// TIA Portal V19 export
DATA_BLOCK "IO-LinkDevicesDB"   // DB210
VERSION : 0.0
// stored: AutoNumber false, InstanceOfName IO-Link Devices, InstanceOfType FB
"IO-Link Devices"
   // VAR
   //    PNIODiag : Struct
   //       StationOK : Bool;
   //       WasUnderMaintenance : Bool;
   //       Maintenance : Bool;
   //       WasFaulty : Bool;
   //       Faulty : Bool;
   //       HadFailed : Bool;
   //       Failed : Bool;
   //       wasDeactivated : Bool;
   //       Deactivated : Bool;
   //    END_STRUCT;
   //    Stat_ReadReq : Bool;
   //    AL2221_100_005_X06 : "IFM_AL2221_PD";
   //    AL2221_100_007_X01 : "IFM_AL2221_PD";
   // END_VAR
BEGIN
END_DATA_BLOCK
